// TIA Portal V14 SP1 export
// export: Created 2019-07-09T07:48:16.0476873Z, ExportSetting WithDefaults, WithReadOnly, DisplayName Totally Integrated Automation Portal, DisplayVersion V14 SP1 Update 6, DisplayName TIA Portal Openness, DisplayVersion V14 SP1 Update 6, DisplayName STEP 7 Professional, DisplayVersion V14 SP1 Update 6, DisplayName WinCC Professional, DisplayVersion V14 SP1 Update 6
FUNCTION_BLOCK "214M_Vibrator"   // FB1002, LAD
{ S7_Optimized_Access := 'FALSE' }
VERSION : 0.1
// stored: AutoNumber false, CodeModifiedDate 2019-07-09T07:45:27.1280754Z, CompileDate 2019-07-09T07:45:27.1261223Z, CreationDate 2019-02-04T08:31:08.0295361Z, InterfaceModifiedDate 2018-10-30T12:28:18.462068Z, IsConsistent true, IsIECCheckEnabled false, IsKnowHowProtected false, ISMultiInstanceCapable true, IsWriteProtected false, LibraryConformanceStatus Warning: The object contains access to global data blocks. Warning: The block contains direct access to inputs, outputs, bit memories, indirect access to the registry or indirect access to external memory areas that are unknown at the time of compilation., ModifiedDate 2019-07-09T07:45:27.1280754Z, ParameterModified 2018-04-23T08:12:12.8650856Z, StructureModified 2018-10-30T12:24:19.5691813Z, UDAEnableTagReadback false
   VAR DB_SPECIFIC
      HMI : Struct
         CMD : Struct
            Start : Bool;   // Команда старта мотора
            Stop : Bool;   // Команда останова вибратора
            Spare_2 : Bool;
            Spare_3 : Bool;
            Spare_4 : Bool;
            Spare_5 : Bool;
            Manual : Bool;   // Ручной режим управления
            Reset_Error : Bool;   // Сброс ошибок
         END_STRUCT;
         DATA : Struct
            StatusWord : Word;   // Слово состояния блока управления мотором
            CntFbkTime : DInt := 1;   // Время контроля включения реле
         END_STRUCT;
      END_STRUCT;
   END_VAR
   VAR
      One_Motor : "OneMotorManag";
   END_VAR
   VAR DB_SPECIFIC
      CntFbkTime : Time;   // Время контроля включения реле
      ResetErr : Bool;   // Сброс ошибок / Dumping of errors of the control package
      General_cond_OK : Bool;   // Готовность электрических систем / Conditions of permission of operation of the mechanism are not satisfied
      ManCmd_StartMov : Bool;   // Старт вращения в ручном режиме / Existence of command for rotation of the motor in manual
      ManCmd_StopMov : Bool;   // Стоп вращения в ручном режиме / Existence of command for a stop of rotation of the motor in manual
      AutoCmd_StartMov : Bool;   // Старт вращения в автоматическом режиме / Existence of command for rotation of the motor in the automatic
      AutoCmd_StopMov : Bool;   // Стоп вращения в автоматическом режиме / Existence of command for a stop of rotation of the motor in the automatic
   END_VAR
   VAR_TEMP
      TempBIT : Bool;   // Command 1 on operation of the mechanism in the automatic mode
   END_VAR
   VAR_TEMP   // added for the SCL form of the ladder/FBD networks
      _w1 : Bool;
   END_VAR
BEGIN

REGION Network 1: Сброс ошибок
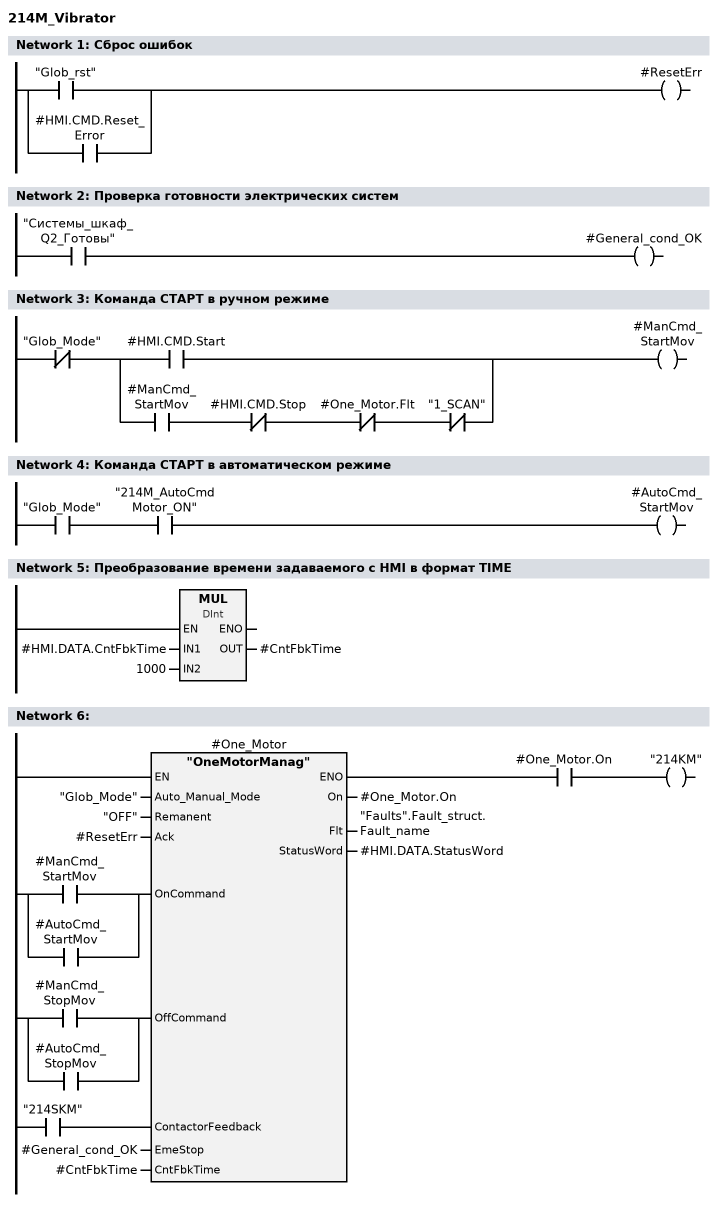
   RUNG wire#powerrail
      Contact( "Glob_rst" )
      wire#w1
      Coil( #ResetErr )
   END_RUNG
   RUNG wire#powerrail
      Contact( #HMI.CMD.Reset_Error )
   END_RUNG wire#w1
   // the same network as SCL:
   #ResetErr := "Glob_rst" OR #HMI.CMD.Reset_Error;
END_REGION

REGION Network 2: Проверка готовности электрических систем
   RUNG wire#powerrail
      Contact( "Системы_шкаф_Q2_Готовы" )
      Coil( #General_cond_OK )
   END_RUNG
   // the same network as SCL:
   #General_cond_OK := "Системы_шкаф_Q2_Готовы";
END_REGION

REGION Network 3: Команда СТАРТ в ручном режиме
   RUNG wire#powerrail
      I_Contact( "Glob_Mode" )
      wire#w1
      Contact( #HMI.CMD.Start )
      wire#w2
      Coil( #ManCmd_StartMov )
   END_RUNG
   RUNG wire#w1
      Contact( #ManCmd_StartMov )
      I_Contact( #HMI.CMD.Stop )
      I_Contact( #One_Motor.Flt )
      I_Contact( "1_SCAN" )
   END_RUNG wire#w2
   // the same network as SCL:
   #ManCmd_StartMov := NOT "Glob_Mode" AND (#HMI.CMD.Start OR (#ManCmd_StartMov AND NOT #HMI.CMD.Stop AND NOT #One_Motor.Flt AND NOT "1_SCAN"));
END_REGION

REGION Network 4: Команда СТАРТ в автоматическом режиме
   RUNG wire#powerrail
      Contact( "Glob_Mode" )
      Contact( "214M_AutoCmdMotor_ON" )
      Coil( #AutoCmd_StartMov )
   END_RUNG
   // the same network as SCL:
   #AutoCmd_StartMov := "Glob_Mode" AND "214M_AutoCmdMotor_ON";
END_REGION

REGION Network 5: Преобразование времени задаваемого с HMI в формат TIME
   RUNG wire#powerrail
      { S7_Templates := "SrcType := DInt"; S7_GenerateENO := "TRUE" } Mul(in1 := #HMI.DATA.CntFbkTime, in2 := 1000, out => #CntFbkTime)
   END_RUNG
   // the same network as SCL:
   #CntFbkTime := #HMI.DATA.CntFbkTime * 1000;
END_REGION

REGION Network 6
   RUNG wire#powerrail
      #One_Motor(OnCommand := wire#w1, OffCommand := wire#w2, ContactorFeedback := wire#w3, Auto_Manual_Mode := "Glob_Mode", Remanent := "OFF", Ack := #ResetErr, EmeStop := #General_cond_OK, CntFbkTime := #CntFbkTime, On => #One_Motor.On, Flt => "Faults".Fault_struct.Fault_name, StatusWord => #HMI.DATA.StatusWord)
      Contact( #One_Motor.On )
      Coil( "214KM" )
   END_RUNG
   RUNG wire#powerrail
      Contact( #ManCmd_StartMov )
   END_RUNG wire#w1
   RUNG wire#powerrail
      Contact( #AutoCmd_StartMov )
   END_RUNG wire#w1
   RUNG wire#powerrail
      Contact( #ManCmd_StopMov )
   END_RUNG wire#w2
   RUNG wire#powerrail
      Contact( #AutoCmd_StopMov )
   END_RUNG wire#w2
   RUNG wire#powerrail
      Contact( "214SKM" )
   END_RUNG wire#w3
   // the same network as SCL:
   #One_Motor(Auto_Manual_Mode := "Glob_Mode",   // "OneMotorManag"
              Remanent := "OFF",
              Ack := #ResetErr,
              OnCommand := #ManCmd_StartMov OR #AutoCmd_StartMov,
              OffCommand := #ManCmd_StopMov OR #AutoCmd_StopMov,
              ContactorFeedback := "214SKM",
              EmeStop := #General_cond_OK,
              CntFbkTime := #CntFbkTime,
              On => #One_Motor.On,
              Flt => "Faults".Fault_struct.Fault_name,
              StatusWord => #HMI.DATA.StatusWord,
              ENO => #_w1);
   "214KM" := #_w1 AND #One_Motor.On;
END_REGION
END_FUNCTION_BLOCK
